(* IEC 61131-3 sources: test/Class/HmiFont35, 1 file *)

(* ---- HmiFont35.st ---- *)
(*!
<Class
	Name               = "HmiFont35"
	Revision           = "0.2"
	RealtimeTask       = "false"
	CyclicTask         = "false"
	BackgroundTask     = "false"
	Sigmatek           = "true"
	OSInterface        = "false"
	HighPriority       = "false"
	Automatic          = "false"
	UpdateMode         = "Prescan"
	SharedCommandTable = "true"
	Objectsize         = "(284,120)">
	<Channels>
		<Server Name="ByteSize" Visualized="false" Initialize="false" WriteProtected="true" Retentive="false"/>
		<Server Name="ClassSvr" Visualized="false" Initialize="false" WriteProtected="true" Retentive="false"/>
		<Client Name="StdLib" Required="false" Internal="false"/>
	</Channels>
	<RevDoku>
		<Owner Company="sigmatek" Author="kolott"/>
		<Dokumentation Revision="0.2" Date="2018-08-31" Author="kolott" Company="sigmatek" Description="cTor added"/>
		<Dokumentation Revision="0.1" Date="2014-03-26" Author="kolott" Company="sigmatek" Description="Innovation: ClassSvr will represent number of used fonts in hmi&#13;&#10;server ByteSize added"/>
	</RevDoku>
</Class>
*)
HmiFont35 : CLASS
  //Servers:
	ClassSvr 	: SvrChCmd_DINT;
	ByteSize 	: SvrCh_UDINT;
  //Clients:
	StdLib 	: CltChCmd__StdLib;
  //Variables:
  //Functions:

	FUNCTION HmiFont35
		VAR_OUTPUT
			ret_code 	: ConfStates;
		END_VAR;

	FUNCTION GLOBAL Free;

	FUNCTION GLOBAL Start;

	FUNCTION GLOBAL CreateList
		VAR_INPUT
			pfnt 	: ^void;
			size 	: UDINT;
		END_VAR
		VAR_OUTPUT
			retcode 	: ^void;
		END_VAR;

	FUNCTION DefaultInit;
  //Tables:
	FUNCTION @STD
		VAR_OUTPUT
			ret_code	: CONFSTATES;
		END_VAR;
	FUNCTION GLOBAL TAB @CT_;
END_CLASS;

#pragma usingLtd _StdLib

#includeC "..\LseEasy\Create.h"

FUNCTION HmiFont35::HmiFont35
	VAR_OUTPUT
		ret_code 	: ConfStates;
	END_VAR

	ret_code := C_OK;
  ByteSize := 0;
  ClassSvr := 0;
  DefaultInit();

END_FUNCTION

FUNCTION HmiFont35::DefaultInit

END_FUNCTION

FUNCTION GLOBAL HmiFont35::Free

  DefaultInit();

END_FUNCTION

FUNCTION GLOBAL HmiFont35::Start

  Free();
  ByteSize := 0;
  ClassSvr := 0;

END_FUNCTION

FUNCTION GLOBAL HmiFont35::CreateList
	VAR_INPUT
		pfnt 	: ^void;
		size 	: udint;
	END_VAR
	VAR_OUTPUT
		retcode 	: ^void;
	END_VAR
  VAR
    pbox : ^_BOX_FONTLIST;
  END_VAR

  retcode := NIL;

  if(pfnt <> NIL) then
    retcode   := StdLib.MallocV1(size + sizeof(_BOX_FONTLIST) - 1, 0);

    if(retcode <> NIL) then
      pbox$^void := retcode;
      _memcpy(#pbox^.data[0], pfnt, size);
      pbox^.boxhdr.size := 0;
      end_BIGBOX_HEADER(#pbox^.boxhdr, size + sizeof(_BOX_FONTLIST) - 1);
      ClassSvr += 1;
      ByteSize += pbox^.boxhdr.size;
    end_if;
  end_if;

END_FUNCTION
